(* CODESYS project cylinders_initial.export

Project tree, tasks and I/O mapping:
  control/
    function block CylinderFB [LD]
    program cylinder_ctrl [LD]
    program cylinder_ctrl_SFC [LD]
    function block LampCTRL [SFC]
    function block Sequence [SFC]
*)

// control/CylinderFB
FUNCTION_BLOCK CylinderFB
VAR_INPUT
	extend: BOOL;	// signal to extend. Extends on positive edge
	retract: BOOL;	// signal to retract
	cyl_in: BOOL;	// sensor that cylinder is not extended, i.e. in
	cyl_out: BOOL;	// sensor that cylinder is not extended, i.e. in
	delay: TIME;
END_VAR
VAR_OUTPUT
	ctrl: BOOL;	// sensor that cylinder is not extended, i.e. in
	count: INT :=0;	// times the cylinder has been extended (cyl_out became true)
END_VAR
VAR
	ton_cyl1: TON;

	ton_cyl23: TON;
	stop: BOOL;
	converstion: BOOL;
	
	t: INT :=5;
END_VAR
VAR // added by the converter: edge detectors and wires of the graphical bodies
    _rt1 : R_TRIG;
END_VAR

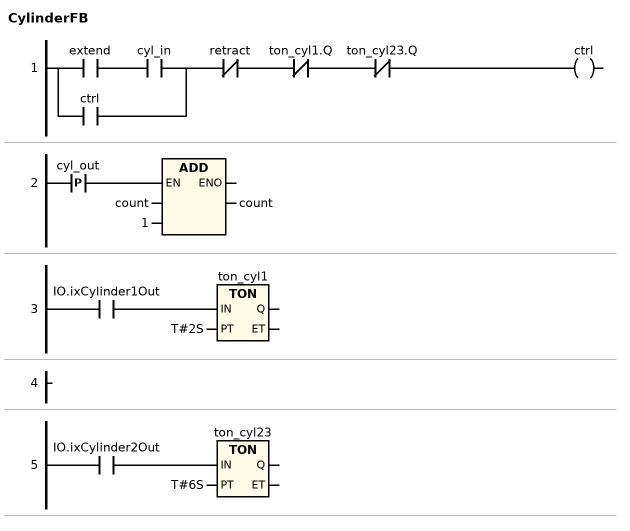
// NETWORK 1
ctrl := (extend AND cyl_in OR ctrl) AND NOT retract AND NOT ton_cyl1.Q AND NOT ton_cyl23.Q;

// NETWORK 2
_rt1(CLK := cyl_out);
IF _rt1.Q THEN count := count + 1; END_IF

// NETWORK 3
ton_cyl1(IN := IO.ixCylinder1Out, PT := T#2S); // TON

// NETWORK 4

// NETWORK 5
ton_cyl23(IN := IO.ixCylinder2Out, PT := T#6S); // TON

END_FUNCTION_BLOCK

// control/cylinder_ctrl
PROGRAM cylinder_ctrl
VAR
	cylinder1: CylinderFB;
	cylinder2: CylinderFB;
	cylinder3: CylinderFB;
	
	init: BOOL := TRUE;
	starting: BOOL;
	cy1_1_out: BOOL;
	cy1_1_done: BOOL;
	
	starting23: BOOL;
	cy1_23_out: BOOL;
	cy1_23_done: BOOL;
		
	LampCTRL_0: LampCTRL;
	lamp_testing: LampCTRL;
END_VAR
VAR // added by the converter: edge detectors and wires of the graphical bodies
    _rt1 : R_TRIG;
    _w1, _w2, _w3, _w4, _w5 : BOOL;
    _ft1 : F_TRIG;
END_VAR

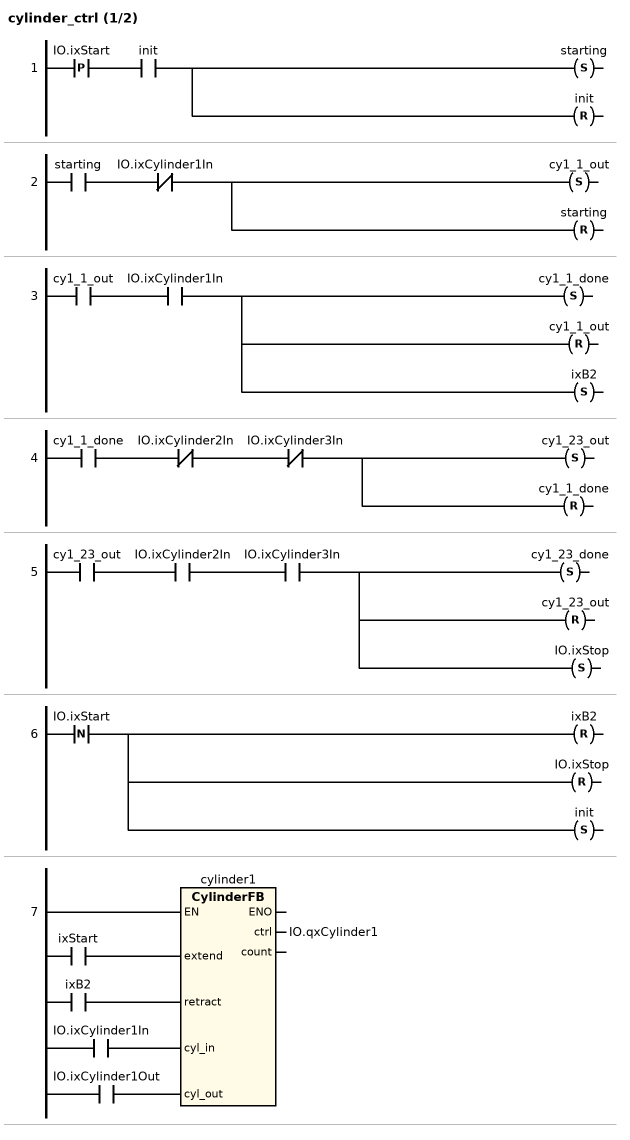
// NETWORK 1
_rt1(CLK := IO.ixStart);
_w1 := _rt1.Q AND init;
starting S= _w1;
init R= _w1;

// NETWORK 2
_w2 := starting AND NOT IO.ixCylinder1In;
cy1_1_out S= _w2;
starting R= _w2;

// NETWORK 3
_w3 := cy1_1_out AND IO.ixCylinder1In;
cy1_1_done S= _w3;
cy1_1_out R= _w3;
ixB2 S= _w3;

// NETWORK 4
_w4 := cy1_1_done AND NOT IO.ixCylinder2In AND NOT IO.ixCylinder3In;
cy1_23_out S= _w4;
cy1_1_done R= _w4;

// NETWORK 5
_w5 := cy1_23_out AND IO.ixCylinder2In AND IO.ixCylinder3In;
cy1_23_done S= _w5;
cy1_23_out R= _w5;
IO.ixStop S= _w5;

// NETWORK 6
_ft1(CLK := IO.ixStart);
ixB2 R= _ft1.Q;
IO.ixStop R= _ft1.Q;
init S= _ft1.Q;

// NETWORK 7
cylinder1(
    extend := ixStart,
    retract := ixB2,
    cyl_in := IO.ixCylinder1In,
    cyl_out := IO.ixCylinder1Out,
    ctrl => IO.qxCylinder1); // CylinderFB

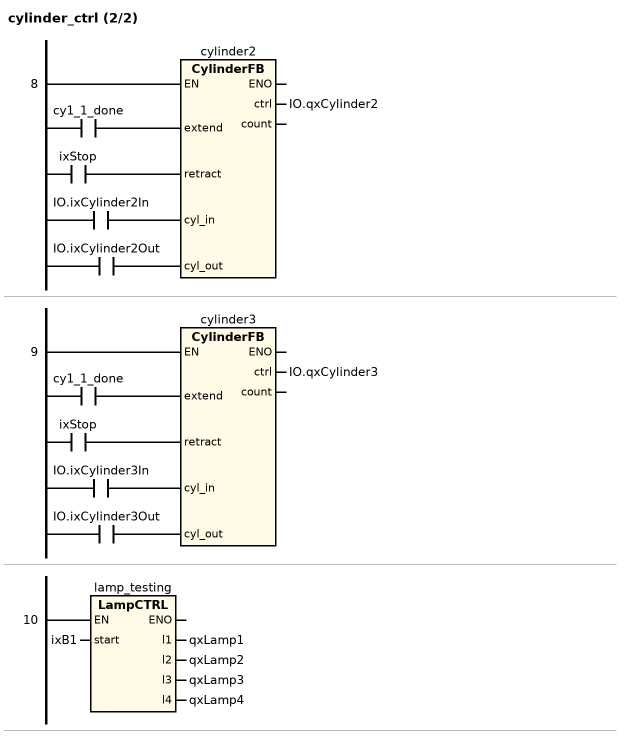
// NETWORK 8
cylinder2(
    extend := cy1_1_done,
    retract := ixStop,
    cyl_in := IO.ixCylinder2In,
    cyl_out := IO.ixCylinder2Out,
    ctrl => IO.qxCylinder2); // CylinderFB

// NETWORK 9
cylinder3(
    extend := cy1_1_done,
    retract := ixStop,
    cyl_in := IO.ixCylinder3In,
    cyl_out := IO.ixCylinder3Out,
    ctrl => IO.qxCylinder3); // CylinderFB

// NETWORK 10
lamp_testing(start := ixB1, l1 => qxLamp1, l2 => qxLamp2, l3 => qxLamp3, l4 => qxLamp4); // LampCTRL

END_PROGRAM

// control/LampCTRL
FUNCTION_BLOCK LampCTRL
VAR_INPUT
	start: BOOL;
END_VAR
VAR_OUTPUT
	l1: BOOL;
	l2: BOOL;
	l3: BOOL;
	l4: BOOL;
END_VAR
VAR
END_VAR

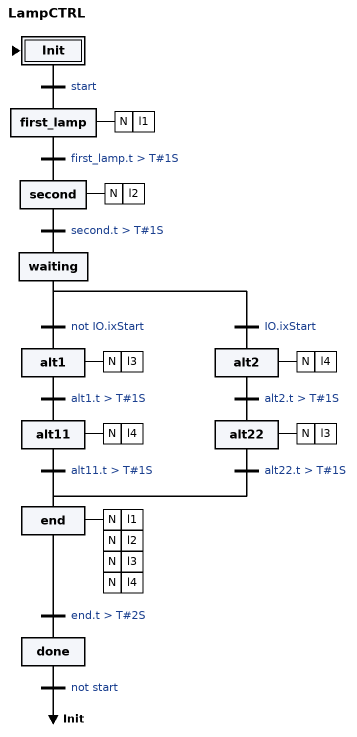
INITIAL_STEP Init:
END_STEP
TRANSITION FROM Init TO first_lamp
    := start;
END_TRANSITION
STEP first_lamp:
    l1(N);
END_STEP
TRANSITION FROM first_lamp TO second
    := first_lamp.t > T#1S;
END_TRANSITION
STEP second:
    l2(N);
END_STEP
TRANSITION FROM second TO waiting
    := second.t > T#1S;
END_TRANSITION
STEP waiting:
END_STEP
TRANSITION FROM waiting TO alt1
    := not IO.ixStart;
END_TRANSITION
STEP alt1:
    l3(N);
END_STEP
TRANSITION FROM alt1 TO alt11
    := alt1.t > T#1S;
END_TRANSITION
STEP alt11:
    l4(N);
END_STEP
TRANSITION FROM alt11 TO end
    := alt11.t > T#1S;
END_TRANSITION
TRANSITION FROM waiting TO alt2
    := IO.ixStart;
END_TRANSITION
STEP alt2:
    l4(N);
END_STEP
TRANSITION FROM alt2 TO alt22
    := alt2.t > T#1S;
END_TRANSITION
STEP alt22:
    l3(N);
END_STEP
TRANSITION FROM alt22 TO end
    := alt22.t > T#1S;
END_TRANSITION
STEP end:
    l1(N);
    l2(N);
    l3(N);
    l4(N);
END_STEP
TRANSITION FROM end TO done
    := end.t > T#2S;
END_TRANSITION
STEP done:
END_STEP
TRANSITION FROM done TO Init
    := not start;
END_TRANSITION

END_FUNCTION_BLOCK

// control/cylinder_ctrl_SFC
PROGRAM cylinder_ctrl_SFC
VAR
	cylinder1: CylinderFB;
	cylinder2: CylinderFB;
	cylinder3: CylinderFB;
	
	sequence_ctrl1: Sequence;
	sequence_ctrl23: Sequence;
	
	LampCTRL_0: LampCTRL;
	lamp_testing: LampCTRL;
END_VAR

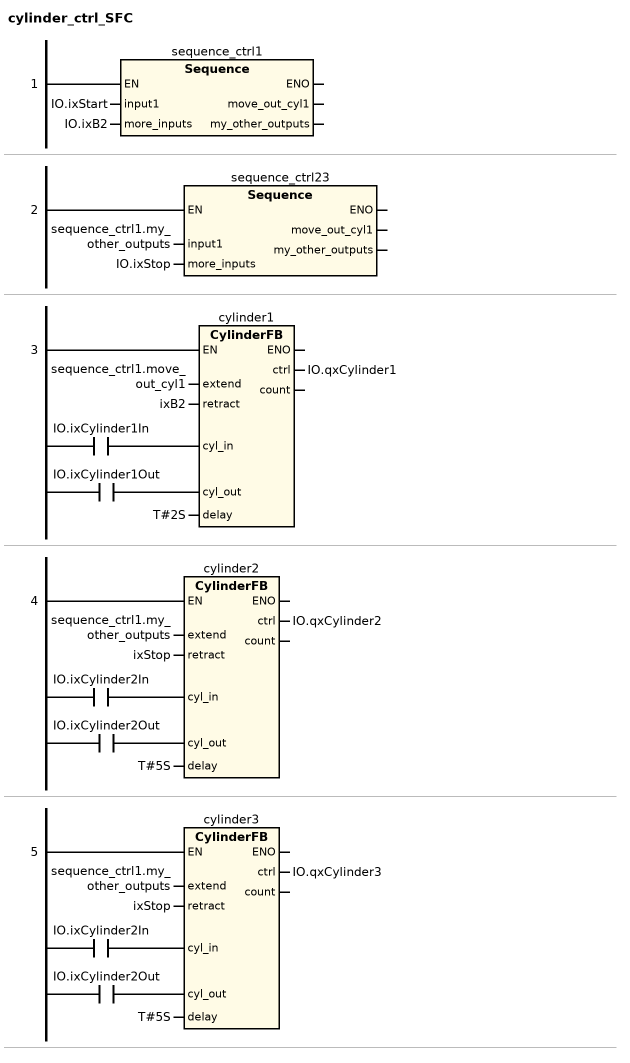
// NETWORK 1
sequence_ctrl1(input1 := IO.ixStart, more_inputs := IO.ixB2); // Sequence

// NETWORK 2
sequence_ctrl23(input1 := sequence_ctrl1.my_other_outputs, more_inputs := IO.ixStop); // Sequence

// NETWORK 3
cylinder1(
    extend := sequence_ctrl1.move_out_cyl1,
    retract := ixB2,
    cyl_in := IO.ixCylinder1In,
    cyl_out := IO.ixCylinder1Out,
    delay := T#2S,
    ctrl => IO.qxCylinder1); // CylinderFB

// NETWORK 4
cylinder2(
    extend := sequence_ctrl1.my_other_outputs,
    retract := ixStop,
    cyl_in := IO.ixCylinder2In,
    cyl_out := IO.ixCylinder2Out,
    delay := T#5S,
    ctrl => IO.qxCylinder2); // CylinderFB

// NETWORK 5
cylinder3(
    extend := sequence_ctrl1.my_other_outputs,
    retract := ixStop,
    cyl_in := IO.ixCylinder2In,
    cyl_out := IO.ixCylinder2Out,
    delay := T#5S,
    ctrl => IO.qxCylinder3); // CylinderFB

END_PROGRAM

// control/Sequence
FUNCTION_BLOCK Sequence
VAR_INPUT
	input1: BOOL;
	more_inputs: BOOL;
END_VAR
VAR_OUTPUT
	move_out_cyl1: BOOL;
	my_other_outputs: BOOL;
END_VAR
VAR
	init: BOOL := TRUE;
END_VAR

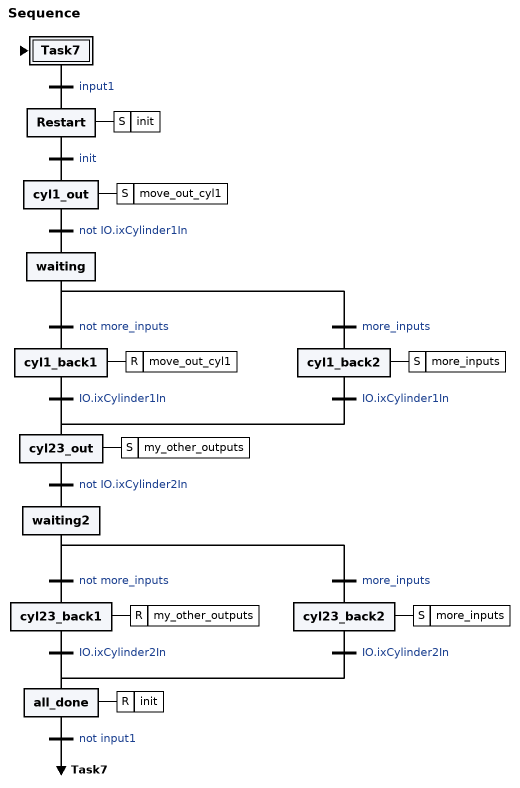
INITIAL_STEP Task7:
END_STEP
TRANSITION FROM Task7 TO Restart
    := input1;
END_TRANSITION
STEP Restart:
    init(S);
END_STEP
TRANSITION FROM Restart TO cyl1_out
    := init;
END_TRANSITION
STEP cyl1_out:
    move_out_cyl1(S);
END_STEP
TRANSITION FROM cyl1_out TO waiting
    := not IO.ixCylinder1In;
END_TRANSITION
STEP waiting:
END_STEP
TRANSITION FROM waiting TO cyl1_back1
    := not more_inputs;
END_TRANSITION
STEP cyl1_back1:
    move_out_cyl1(R);
END_STEP
TRANSITION FROM cyl1_back1 TO cyl23_out
    := IO.ixCylinder1In;
END_TRANSITION
TRANSITION FROM waiting TO cyl1_back2
    := more_inputs;
END_TRANSITION
STEP cyl1_back2:
    more_inputs(S);
END_STEP
TRANSITION FROM cyl1_back2 TO cyl23_out
    := IO.ixCylinder1In;
END_TRANSITION
STEP cyl23_out:
    my_other_outputs(S);
END_STEP
TRANSITION FROM cyl23_out TO waiting2
    := not IO.ixCylinder2In;
END_TRANSITION
STEP waiting2:
END_STEP
TRANSITION FROM waiting2 TO cyl23_back1
    := not more_inputs;
END_TRANSITION
STEP cyl23_back1:
    my_other_outputs(R);
END_STEP
TRANSITION FROM cyl23_back1 TO all_done
    := IO.ixCylinder2In;
END_TRANSITION
TRANSITION FROM waiting2 TO cyl23_back2
    := more_inputs;
END_TRANSITION
STEP cyl23_back2:
    more_inputs(S);
END_STEP
TRANSITION FROM cyl23_back2 TO all_done
    := IO.ixCylinder2In;
END_TRANSITION
STEP all_done:
    init(R);
END_STEP
TRANSITION FROM all_done TO Task7
    := not input1;
END_TRANSITION

END_FUNCTION_BLOCK
